{attribute addProperty BoxType "EL3773-0000-0018"}
{attribute addProperty Id "I2_SamplesAT %I*ARRAY [1..10] OF INT16020"}
{attribute addProperty CRC "3414361115"}
{attribute addProperty SizeInBites "160"}
{attribute addProperty SizeInBytes "20"}
TYPE L2_Current_Samples_CB83041B :
STRUCT
	{attribute addProperty Name "I2_Samples"}
	I2_Samples AT %I* : ARRAY [1..10] OF INT;
END_STRUCT
END_TYPE

(* stored: Version 1.2.0.0, ProductVersion 3.1.4024.9
   DUT L2_Current_Samples_CB83041B: Id {330dd16a-aeab-4636-80a8-f53b1d228f00} *)
